{attribute 'qualified_only'}
{attribute 'strict'}
TYPE E_IOElectrovalveType :
(
	NC_3na2 	:= 0,
	NO_3na2		:= 1,
	C1_5na2		:= 2,
	C2_5na2		:= 3,
	C2_5na3O	:= 4,	//odpowietrzony
	C2_5na3Z	:= 5	//Zapowietrzony
);
END_TYPE

(* stored: Version 1.1.0.1
   DUT E_IOElectrovalveType: Id {77395edc-00f8-4838-aa63-45bee668a694} *)
